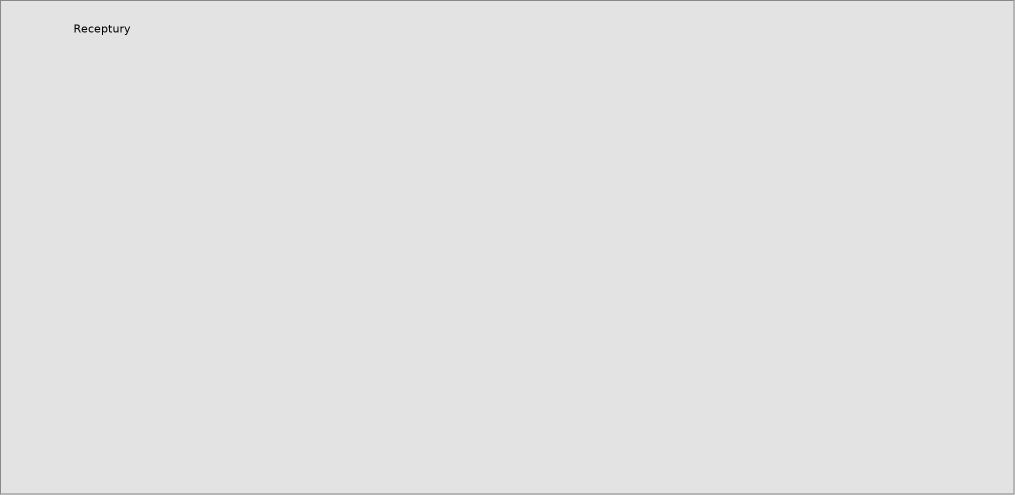
VISUALIZATION F_02_Recipe  // 1015x495
VAR_IN_OUT
	stScreenData	: ST_MCHMIPrepareScreen_02_XX;
	
END_VAR
    Label (27,14 150x30), "Receptury"
END_VISUALIZATION

(* stored: Version 1.1.0.1
   Visu F_02_Recipe: Id {64ca99b3-9e34-0291-2f42-b48227333204} *)
